FUNCTION_BLOCK CSVWRITER_-2120031061
  (* Standard: 61499-2 *)
  (* Version 1.0, 2010-03-25, stano, nxtControl GmbH, template *)
  PACKAGE Main;
  (* Compiler Cpp *)
  {SET_ATTRIBUTE(Runtime.FBType.ImplementingType, nxtControl.Standard#DYNGEN_CSVWRITER)}
  {SET_ATTRIBUTE(Configuration.GenericFBType.InterfaceParams, nxtControl.Standard#I:=3;data${I$}:STRING,STRING,STRING)}
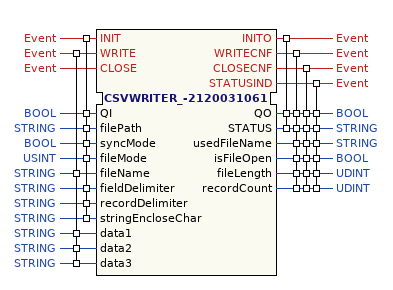
  EVENT_INPUT
    INIT WITH QI, filePath, syncMode, fileMode, fieldDelimiter, recordDelimiter, stringEncloseChar;
    WRITE WITH fileName, data1, data2, data3; (* Write a record into the current file (open if necessary) *)
    CLOSE; (* Closes the current file *)
  END_EVENT
  EVENT_OUTPUT
    INITO WITH QO, STATUS;
    WRITECNF WITH QO, STATUS, usedFileName, isFileOpen, fileLength, recordCount; (* Confirms queuing the data for writing. Does not mean the data were actually written into the file *)
    CLOSECNF WITH QO, STATUS, usedFileName, isFileOpen, fileLength, recordCount; (* Confirms closing of the current file *)
    STATUSIND WITH QO, STATUS, usedFileName, isFileOpen, fileLength, recordCount; (* Indicates change of the file status *)
  END_EVENT
  VAR_INPUT
    QI : BOOL;
    filePath : STRING; (* Path of the destination file, relative to appdata or in config specified root *)
    syncMode : BOOL; (* Flush the file after each write operation *)
    fileMode : USINT; {SET_ATTRIBUTE(ParameterEditor, ComboBox{Enums=APPEND = 0|OVERWRITE = 1$})}
    fileName : STRING; (* Name of the destination file *)
    fieldDelimiter : STRING; (* String delimiting the values (\t possible) *)
    recordDelimiter : STRING; (* String delimiting the records (\r, \n possible) *)
    stringEncloseChar : STRING; (* String enclosing character (or empty for no enclosing) *)
    data1 : STRING; (* Data to write *)
    data2 : STRING; (* Data to write *)
    data3 : STRING; (* Data to write *)
  END_VAR
  VAR_OUTPUT
    QO : BOOL;
    STATUS : STRING;
    usedFileName : STRING; (* Name of the file currently used for writing *)
    isFileOpen : BOOL; (* Open status *)
    fileLength : UDINT; (* Current length of the file *)
    recordCount : UDINT; (* Number of the records written since last file open *)
  END_VAR
  EC_STATES
    START;
  END_STATES
END_FUNCTION_BLOCK
